(* CODESYS project AM402.project

Project tree, tasks and I/O mapping:
  Device : AM402-CPU1608TP/TN, Shenzhen Inovance Control Technology, version 3.5.11.11
    application Application
      libraries: Standard, * (System); SysTimeRtc, * (System); CmpHCMotion, 1.1.0.2 (Inovance); MemoryUtils, * (3S - Smart Software Solutions GmbH)
      task ETHERCAT (cyclic, interval 4000 µs, priority 0) calls ETHERCAT.EtherCAT_Task, MAIN
      program MAIN [ST]: io, motion, save_check, save_apply, supply, work, cut, cut_profile_update
      DataMain/
        data type HMIData
        data type SaveData
        data type SaveDataBig
        data type ProcessData
      DataWork/
        data type SupplyData
        data type WorkData
        data type CutData
        data type CutProfile
        data type CutProfileStep
      Enum/
        data type State
      Object/
        data type Button
        data type Cylinder
        data type AxisLinear
      function StateNext [ST]
      Symbols
      function block AxisLinearFB [ST]
    HardWare Configuration
    Network Configuration
      LocalBus Config
      EtherCAT Config
    Device Diagnosis
    Resources List
    ConfigStorage
    SoftMotion General Axis Pool
    HIGH_SPEED_IO : High Speed IO Module, Inovance, version 00.00.00.20
        unmapped channels: InputData, OutputData
      HSIO
    HwConfiguratioinDevice : SystemHardwareConfig, AM600 of Inovance, version 00.00.00.10
        settings: NetworkConfigArray.NetworkConfigArray.BusType = 10; NetworkConfigArray.NetworkConfigArray.RackSum = 1; NetworkConfigArray.NetworkConfigArray.HardwareConfigArray.HardwareConfigArray.RackNo = 1
    ETHERCAT : EtherCAT Master SoftMotion, 3S - Smart Software Solutions GmbH, version 3.5.11.10
        settings:  = 0; NetworkName = 'eth1'; SelectNetworkByName = TRUE; DisableTaskGeneration = True; SyncOffset = 20
      XINJE_DS5C1_CoE_Drive_Rev4_0 : XINJE-DS5C1 EtherCAT(CoE) Drive Rev4.0 v3.7.70, Xinje Electronics, Inc., order no. XINJE-DS5C1 CoE Drive Rev4.0, version Revision=16#20201207
          settings: StationAlias = 1; DC sync0 cycletime = 4000; DC sync1 cycletime = 4000; Interpolation time period.Value = 4
          unmapped channels: Control Word, TargetPosition, TargetVelocity, TargetTorque, ModeOfOperation, Status Word, ActualPosition, Velocity actual value, ActualTorque, ModeOfOperationDisplay
        Axis : Axis, 3S - Smart Software Solutions GmbH, order no. 0, version 4.0.0.0
            settings: wDriveID = 0; dwRatioTechUnitsDenom = 16384; iRatioTechUnitsNum = 625; eRampType = 3; ScalingIncs = 131072; ScalingUnits = 5000; AdrOffset_8010 = 2; BitOffset_8010 = 0; BitLength_8010 = 16; Address_8010 = '%QW1'; Type_8010 = 'UINT'; AddressPointer_8010 = ADR(%QW1); AdrOffset_8020 = 4; BitOffset_8020 = 0; BitLength_8020 = 32; Address_8020 = '%QD1'; Type_8020 = 'DINT'; AddressPointer_8020 = ADR(%QD1); AdrOffset_8030 = 8; BitOffset_8030 = 0; BitLength_8030 = 32; Address_8030 = '%QD2'; Type_8030 = 'DINT'; AddressPointer_8030 = ADR(%QD2); AdrOffset_8040 = 12; BitOffset_8040 = 0; BitLength_8040 = 16; Address_8040 = '%QW6'; Type_8040 = 'INT'; AddressPointer_8040 = ADR(%QW6); AdrOffset_8050 = 14; BitOffset_8050 = 0; BitLength_8050 = 8; Address_8050 = '%QB14'; Type_8050 = 'SINT'; AddressPointer_8050 = ADR(%QB14); AdrOffset_8060 = 4294967295; BitOffset_8060 = 0; BitLength_8060 = 0; Address_8060 = '';
              Type_8060 = ''; AddressPointer_8060 = 0; AdrOffset_8070 = 4294967295; BitOffset_8070 = 0; BitLength_8070 = 0; Address_8070 = ''; Type_8070 = ''; AddressPointer_8070 = 0; AdrOffset_8080 = 4294967295; BitOffset_8080 = 0; BitLength_8080 = 0; Address_8080 = ''; Type_8080 = ''; AddressPointer_8080 = 0; AdrOffset_8090 = 4294967295; BitOffset_8090 = 0; BitLength_8090 = 0; Address_8090 = ''; Type_8090 = ''; AddressPointer_8090 = 0; AdrOffset_8100 = 4294967295; BitOffset_8100 = 0; BitLength_8100 = 0; Address_8100 = ''; Type_8100 = ''; AddressPointer_8100 = 0; AdrOffset_8510 = 2; BitOffset_8510 = 0; BitLength_8510 = 16; Address_8510 = '%IW1'; Type_8510 = 'UINT'; AddressPointer_8510 = ADR(%IW1); AdrOffset_8520 = 4; BitOffset_8520 = 0; BitLength_8520 = 32; Address_8520 = '%ID1'; Type_8520 = 'DINT'; AddressPointer_8520 = ADR(%ID1); AdrOffset_8530 = 8; BitOffset_8530 = 0;
              BitLength_8530 = 32; Address_8530 = '%ID2'; Type_8530 = 'DINT'; AddressPointer_8530 = ADR(%ID2); AdrOffset_8540 = 12; BitOffset_8540 = 0; BitLength_8540 = 16; Address_8540 = '%IW6'; Type_8540 = 'INT'; AddressPointer_8540 = ADR(%IW6); AdrOffset_8550 = 14; BitOffset_8550 = 0; BitLength_8550 = 8; Address_8550 = '%IB14'; Type_8550 = 'SINT'; AddressPointer_8550 = ADR(%IB14); AdrOffset_8560 = 4294967295; BitOffset_8560 = 0; BitLength_8560 = 0; Address_8560 = ''; Type_8560 = ''; AddressPointer_8560 = 0; AdrOffset_8570 = 4294967295; BitOffset_8570 = 0; BitLength_8570 = 0; Address_8570 = ''; Type_8570 = ''; AddressPointer_8570 = 0; AdrOffset_8580 = 4294967295; BitOffset_8580 = 0; BitLength_8580 = 0; Address_8580 = ''; Type_8580 = ''; AddressPointer_8580 = 0; AdrOffset_8590 = 4294967295; BitOffset_8590 = 0; BitLength_8590 = 0; Address_8590 = ''; Type_8590 = ''; AddressPointer_8590 = 0;
              AdrOffset_8600 = 4294967295; BitOffset_8600 = 0; BitLength_8600 = 0; Address_8600 = ''; Type_8600 = ''; AddressPointer_8600 = 0; AdrOffset_8600 = 4294967295; BitOffset_8600 = 0; BitLength_8600 = 0; Address_8610 = ''; Type_8610 = ''; AddressPointer_8610 = 0; AdrOffset_8620 = 4294967295; BitOffset_8620 = 0; BitLength_8620 = 0; Address_8620 = ''; Type_8620 = ''; AddressPointer_8620 = 0
      XINJE_DS5C1_CoE_Drive_Rev4_0_1 : XINJE-DS5C1 EtherCAT(CoE) Drive Rev4.0 v3.7.70, Xinje Electronics, Inc., order no. XINJE-DS5C1 CoE Drive Rev4.0, version Revision=16#20201207
          settings: StationAlias = 1; DC sync0 cycletime = 4000; DC sync1 cycletime = 4000; Interpolation time period.Value = 4
          unmapped channels: Control Word, TargetPosition, TargetVelocity, TargetTorque, ModeOfOperation, Status Word, ActualPosition, Velocity actual value, ActualTorque, ModeOfOperationDisplay
        Axis_1 : Axis, 3S - Smart Software Solutions GmbH, order no. 0, version 4.0.0.0
            settings: dwRatioTechUnitsDenom = 16384; iRatioTechUnitsNum = -625; eRampType = 3; ScalingIncs = 131072; ScalingUnits = 5000; InvertDirection = TRUE; AdrOffset_8010 = 16; BitOffset_8010 = 0; BitLength_8010 = 16; Address_8010 = '%QW8'; Type_8010 = 'UINT'; AddressPointer_8010 = ADR(%QW8); AdrOffset_8020 = 20; BitOffset_8020 = 0; BitLength_8020 = 32; Address_8020 = '%QD5'; Type_8020 = 'DINT'; AddressPointer_8020 = ADR(%QD5); AdrOffset_8030 = 24; BitOffset_8030 = 0; BitLength_8030 = 32; Address_8030 = '%QD6'; Type_8030 = 'DINT'; AddressPointer_8030 = ADR(%QD6); AdrOffset_8040 = 28; BitOffset_8040 = 0; BitLength_8040 = 16; Address_8040 = '%QW14'; Type_8040 = 'INT'; AddressPointer_8040 = ADR(%QW14); AdrOffset_8050 = 30; BitOffset_8050 = 0; BitLength_8050 = 8; Address_8050 = '%QB30'; Type_8050 = 'SINT'; AddressPointer_8050 = ADR(%QB30); AdrOffset_8060 = 4294967295; BitOffset_8060 = 0; BitLength_8060 = 0; Address_8060 = '';
              Type_8060 = ''; AddressPointer_8060 = 0; AdrOffset_8070 = 4294967295; BitOffset_8070 = 0; BitLength_8070 = 0; Address_8070 = ''; Type_8070 = ''; AddressPointer_8070 = 0; AdrOffset_8080 = 4294967295; BitOffset_8080 = 0; BitLength_8080 = 0; Address_8080 = ''; Type_8080 = ''; AddressPointer_8080 = 0; AdrOffset_8090 = 4294967295; BitOffset_8090 = 0; BitLength_8090 = 0; Address_8090 = ''; Type_8090 = ''; AddressPointer_8090 = 0; AdrOffset_8100 = 4294967295; BitOffset_8100 = 0; BitLength_8100 = 0; Address_8100 = ''; Type_8100 = ''; AddressPointer_8100 = 0; AdrOffset_8510 = 16; BitOffset_8510 = 0; BitLength_8510 = 16; Address_8510 = '%IW8'; Type_8510 = 'UINT'; AddressPointer_8510 = ADR(%IW8); AdrOffset_8520 = 20; BitOffset_8520 = 0; BitLength_8520 = 32; Address_8520 = '%ID5'; Type_8520 = 'DINT'; AddressPointer_8520 = ADR(%ID5); AdrOffset_8530 = 24; BitOffset_8530 = 0;
              BitLength_8530 = 32; Address_8530 = '%ID6'; Type_8530 = 'DINT'; AddressPointer_8530 = ADR(%ID6); AdrOffset_8540 = 28; BitOffset_8540 = 0; BitLength_8540 = 16; Address_8540 = '%IW14'; Type_8540 = 'INT'; AddressPointer_8540 = ADR(%IW14); AdrOffset_8550 = 30; BitOffset_8550 = 0; BitLength_8550 = 8; Address_8550 = '%IB30'; Type_8550 = 'SINT'; AddressPointer_8550 = ADR(%IB30); AdrOffset_8560 = 4294967295; BitOffset_8560 = 0; BitLength_8560 = 0; Address_8560 = ''; Type_8560 = ''; AddressPointer_8560 = 0; AdrOffset_8570 = 4294967295; BitOffset_8570 = 0; BitLength_8570 = 0; Address_8570 = ''; Type_8570 = ''; AddressPointer_8570 = 0; AdrOffset_8580 = 4294967295; BitOffset_8580 = 0; BitLength_8580 = 0; Address_8580 = ''; Type_8580 = ''; AddressPointer_8580 = 0; AdrOffset_8590 = 4294967295; BitOffset_8590 = 0; BitLength_8590 = 0; Address_8590 = ''; Type_8590 = ''; AddressPointer_8590 = 0;
              AdrOffset_8600 = 4294967295; BitOffset_8600 = 0; BitLength_8600 = 0; Address_8600 = ''; Type_8600 = ''; AddressPointer_8600 = 0; AdrOffset_8600 = 4294967295; BitOffset_8600 = 0; BitLength_8600 = 0; Address_8610 = ''; Type_8610 = ''; AddressPointer_8610 = 0; AdrOffset_8620 = 4294967295; BitOffset_8620 = 0; BitLength_8620 = 0; Address_8620 = ''; Type_8620 = ''; AddressPointer_8620 = 0
  SMElement/
    SM0_SM511
    SM512_SM1023
    SM1024_SM1535
    SM1536_SM2047
    SM2048_SM2559
    SM2560_SM3071
    SM3072_SM3583
    SM3584_SM4095
    SM4096_SM4607
    SM4608_SM5119
    SM5120_SM5631
    SM5632_SM6143
    SM6144_SM6655
    SM6656_SM7167
    SM7168_SM7679
    SM7680_SM8191
    SM8192_SM8703
    SM8704_SM9215
    SM9216_SM9727
    SM9728_SM9999
  SDElement/
    SD0_SD511
    SD512_SD1023
    SD1024_SD1535
    SD1536_SD2047
    SD2048_SD2559
    SD2560_SD3071
    SD3072_SD3583
    SD3584_SD4095
    SD4096_SD4607
    SD4608_SD5119
    SD5120_SD5631
    SD5632_SD6143
    SD6144_SD6655
    SD6656_SD7167
    SD7168_SD7679
    SD7680_SD8191
    SD8192_SD8703
    SD8704_SD9215
    SD9216_SD9727
    SD9728_SD9999
*)

// Device/Application/DataMain/HMIData
{ attribute 'pack_mode' := ''}
TYPE HMIData :
STRUCT
	//
	save_data: SaveData;
	save: BOOL;
	save_need_check: BOOL;
	save_need: BOOL;
	//
	cut_profile_name_as_array: ARRAY[0..19] OF BYTE;
	cut_profile: CutProfile;
	cut_profile_points_x: ARRAY[0..(5*4-1+4)] OF UDINT;
	cut_profile_points_y: ARRAY[0..(5*4-1+4)] OF UDINT;
	cut_profile_point_count: UINT;
	cut_profile_bound_x: UDINT;
	cut_profile_bound_y: UDINT;
	cut_profile_index_changed: BOOL;
	cut_profile_list_update: BOOL;
	cut_profile_update: BOOL;
	//
	plc_ready: BOOL;
	hmi_ready: BOOL;
	run: BOOL;
	stop: BOOL;
	home: BOOL;
	manual_cut: BOOL;
	//
	supply_clamp_drag: BOOL;
	supply_clamp_hold: BOOL;
	supply_air_cool: BOOL;
	jog_micron_per_sec: UINT;
	jog_n: BOOL;
	jog_p: BOOL;
	jog_index: UINT;
	overload_resolved: BOOL;
	work_piece_count: UINT;
	//
	view_run: BOOL;
	view_stop: BOOL;
	view_air_ready: BOOL;
	view_can_run: BOOL;
	view_can_stop: BOOL;
	view_can_home: BOOL;
	//
	view_supply_position_micron: UDINT;
	view_supply_torque_mNm: UDINT;
	view_supply_foil_position_micron: UDINT;
	view_supply_sensor_hold: BOOL;
	view_supply_sensor_drag: BOOL;
	view_supply_foil_short: BOOL;
	view_cut_position_micron: UDINT;
	view_cut_torque_mNm: UDINT;
	view_cut_depth_micron: UDINT;
	view_work_piece_remain: UINT;
	//
	view_overload: BOOL;
	view_cycle_time_msec: UDINT;
	//
	view_state_work: INT;
	view_state_supply: INT;
	view_state_cut: INT;
END_STRUCT
END_TYPE

// Device/Application/DataMain/SaveData
{ attribute 'pack_mode' := ''}
TYPE SaveData :
STRUCT
	set_done: BOOL;
	//
	supply_ramp_time_msec: UINT;
	supply_jerk_factor: UINT;
	supply_hold_n_delay_msec: UINT;
	supply_hold_p_delay_msec: UINT;
	supply_drag_n_delay_msec: UINT;
	supply_drag_p_delay_msec: UINT;
	//
	cut_ramp_time_msec: UINT;
	cut_jerk_factor: UINT;
	cut_begin_micron: UDINT;
	//
	blade_thickness_micron: UINT; // độ dày lưỡi dao
	cut_depth_end_micron: UDINT; // độ sâu cắt đứt
	cut_retract_micron_per_sec: UDINT; // tốc độ lùi sau khi cắt
	cut_profile_index: UINT;
	manual_cut_micron_per_sec: UDINT; // tốc độ cắt thủ công
	//
	cut_profiles_name: ARRAY[0..9] OF STRING(20);
END_STRUCT
END_TYPE

// Device/Application/DataWork/SupplyData
{ attribute 'pack_mode' := ''}
TYPE SupplyData :
STRUCT
	state: INT;
	sensor_hold: BOOL;
	sensor_drag: BOOL;
	axis: AxisLinear;
	axis_fb: AxisLinearFB;
	clamp_drag: Cylinder;
	clamp_hold: Cylinder;
	air_cool: Cylinder;
	//
	foil_position_micron: LREAL;
	foil_position_target_micron: LREAL;
	foil_micron_per_sec: LREAL;
	foil_position_delta_micron: LREAL;
	foil_short: BOOL;
END_STRUCT
END_TYPE

// Device/Application/DataWork/WorkData
{ attribute 'pack_mode' := ''}
TYPE WorkData :
STRUCT
	state: INT;
	run: Button;
	run_timer: TON;
	can_run: BOOL;
	stop: Button;
	can_stop: BOOL;
	air_ready: BOOL;
	home: Button;
	can_home: BOOL;
	overload: Button;
	jog_i: POINTER TO AxisLinear;
	cut_profile: CutProfile;
	cut_profile_step_index: UINT;
	cut_profile_step: POINTER TO CutProfileStep;
	blade_thickness_micron: LREAL;
	cut_depth_end_micron: LREAL;
	work_piece_remain: UINT;
	manual_cut_clamp: BOOL;
	manual_cut_micron_per_sec: LREAL;
END_STRUCT
END_TYPE

// Device/Application/DataWork/CutData
{ attribute 'pack_mode' := ''}
TYPE CutData :
STRUCT
	state: INT;
	axis: AxisLinear;
	axis_fb: AxisLinearFB;
	blade_is_on: BOOL;
	//
	begin_micron: LREAL;
	depth_micron: LREAL;
	cut_micron_per_sec: LREAL;
	cut_retract_micron_per_sec: LREAL;
END_STRUCT
END_TYPE

// Device/Application/Enum/State
{attribute 'qualified_only'}
{attribute 'strict'}
TYPE State :
(
	NONE := 0,
	RST := 1,
	RST_DONE := 50,
	HOME := 51,
	HOME_FORWARD := 71,
	HOME_DONE := 90,
	HOME_OFFSET := 91,
	HOME_OFFSET_DONE := 99,
	READY := 100,
	RUN := 101,
	RUN_ING := 200
);
END_TYPE

// Device/Application/Object/Button
{ attribute 'pack_mode' := ''}
TYPE Button :
STRUCT
	on: BOOL;
	rise: R_TRIG;
	rise_physical: R_TRIG;
	fall: F_TRIG;
	fall_physical: F_TRIG;
END_STRUCT
END_TYPE

// Device/Application/Object/Cylinder
{ attribute 'pack_mode' := ''}
TYPE Cylinder :
STRUCT
	on: BOOL;
	n_timer: TON;
	p_timer: TON;
END_STRUCT
END_TYPE

// Device/Application/Object/AxisLinear
{ attribute 'pack_mode' := ''}
TYPE AxisLinear :
STRUCT
	///////
	//REF//
	///////
	ref: POINTER TO SM3_Drive_ETC_DS402_CyclicSync.AXIS_REF_ETC_DS402_CS;
	read_status: POINTER TO MC_ReadStatus;
	set_mode: POINTER TO SMC_SetControllerMode;
	limit_torque: POINTER TO MC_SetTorqueLimit;
	power: POINTER TO MC_Power;
	reset: POINTER TO MC_Reset;
	stop: POINTER TO MC_Stop;
	inch: POINTER TO SMC_Inch;
	sp: POINTER TO MC_SetPosition;
	mabs: POINTER TO MC_MoveAbsolute;
	////////
	//DATA//
	////////
	encoder_resolution: UDINT;
	torque_rated_Nm: LREAL;
	///////////
	//PROCESS//
	///////////
	state: INT;
	torque_Nm: LREAL;
	overload: BOOL;
	overload_timer: TON;
	//home
	home_done: BOOL; // = TRUE khi về gốc thành công, chỉ về gốc khi bật máy
	home_torque_Nm: LREAL;
	home_hit_timer: TON;
	home_offset_absolute_micron: LREAL; // vị trí từ điểm va chạm đến gốc tuyệt đối, xem hàm save_apply()
	home_back_micron_per_sec: LREAL; // tốc độ lùi về lấy gốc
	home_forward_micron_per_sec: LREAL; // tốc độ tiến sau khi lấy gốc xong
	home_offset_micron: LREAL; // giá trị này để thực hiện lệnh state = State.HOME_OFFSET ở trong AxisLinearFB
	//
	jog_micron_per_sec: LREAL; // tốc độ jog
	jog_direction: INT; // hướng jog
	max_micron: LREAL; // giới hạn vị trí tối đa có thể di chuyển từ gốc tuyệt đối
	max_micron_per_sec: LREAL; // giới hạn tốc độ tối đa
	ramp_time_sec: LREAL; // thời gian tăng, giảm tốc
	jerk_factor: LREAL; // độ giật, giá trị jerk của các hàm dịch chuyển sẽ bằng jerk := jerk_factor * acceleration
	//run
	target_position_micron: LREAL; // sử dụng cho state = State.RUN ở trong AxisLinearFB
	target_velocity_micron_per_sec: LREAL; // sử dụng cho state = State.RUN ở trong AxisLinearFB
END_STRUCT
END_TYPE

// Device/Application/DataWork/CutProfile
{ attribute 'pack_mode' := ''}
TYPE CutProfile :
STRUCT
	length_micron: UDINT;
	cut_micron_per_sec: UDINT;
	supply_micron_per_sec: UDINT;
	steps: ARRAY[0..4] OF CutProfileStep;
END_STRUCT
END_TYPE

// Device/Application/DataWork/CutProfileStep
{ attribute 'pack_mode' := ''}
TYPE CutProfileStep :
STRUCT
	active: BOOL;
	begin_micron: UDINT;
	width_micron: UDINT;
	depth_begin_micron: UDINT;
	depth_end_micron: UDINT;
END_STRUCT
END_TYPE

// Device/Application/DataMain/SaveDataBig
{ attribute 'pack_mode' := ''}
TYPE SaveDataBig :
STRUCT
	set_done: BOOL;
	//
	cut_profiles: ARRAY[0..9] OF CutProfile;
END_STRUCT
END_TYPE

// Device/Application/DataMain/ProcessData
{ attribute 'pack_mode' := ''}
TYPE ProcessData :
STRUCT
	cut_profile_name: STRING(20);
	cut_profile_name_changed: BOOL;
	cut_profile_changed: BOOL;
	cut_profile_list_update_need: BOOL;
	cut_profile_update_need: BOOL;
	supply_foil_short_rise: R_TRIG;
END_STRUCT
END_TYPE

// Device/Application/MAIN
PROGRAM MAIN
VAR
	RTC_last: ULINT;
	RTC : ULINT;
	//
	axiss: ARRAY [0..1] OF POINTER TO SM3_Drive_ETC_DS402_CyclicSync.AXIS_REF_ETC_DS402_CS;
	// dùng pointer để dễ dàng thao tác với nhiều trục hơn, xem hàm motion()
	axiss_read: ARRAY[0..1] OF SMC3_ETC_ReadParameter_CoE;
	axiss_read_status: ARRAY[0..1] OF MC_ReadStatus;
	axiss_set_mode: ARRAY[0..1] OF SMC_SetControllerMode;
	axiss_limit_torque: ARRAY[0..1] OF MC_SetTorqueLimit; // không có sẵn, cần cài thư viện CmpHCMotion của Inovance, PLC khác có thể khác
	axiss_power: ARRAY[0..1] OF MC_Power; // bật tắt động cơ
	axiss_reset: ARRAY[0..1] OF MC_Reset; // reset lỗi
	axiss_stop: ARRAY[0..1] OF MC_Stop; // dừng
	axiss_inch: ARRAY[0..1] OF SMC_Inch;
	axiss_sp: ARRAY[0..1] OF MC_SetPosition;
	axiss_mabs: ARRAY[0..1] OF MC_MoveAbsolute;
	axiss_encoder_resolution: ARRAY[0..1] OF UDINT;
	axiss_rated_torque_Nm: ARRAY[0..1] OF LREAL;
	axiss_ready: BOOL;
	//
	state_main: INT;
	main_save: Button;
	supply_data: SupplyData;
	cut_data: CutData;
	work_data: WorkData;
	hmi_data: HMIData;
	process_data: ProcessData;
	//
	i: UINT;
	j: UINT;
	k: UINT;
	axis_linear_i: POINTER TO AxisLinear;
	axis_linear_fb_i: POINTER TO AxisLinearFB;
	cut_profile_i: POINTER TO CutProfile;
	cut_profile_step_i: POINTER TO CutProfileStep;
	//
	udint_min: UDINT;
	udint_max: UDINT;
END_VAR

VAR CONSTANT
	c_axis_count: UINT := 2;
	c_axis_i_max: UINT := c_axis_count - 1;
	c_cut_profile_count: UINT := 10;
	c_cut_profile_i_max: UINT := c_cut_profile_count - 1;
	c_cut_profile_step_count: UINT := 5;
	c_cut_profile_step_i_max: UINT := c_cut_profile_step_count - 1;
	c_name_length: UINT := 20;
	c_supply_travel_micron_max: UDINT := 289_000;
	c_supply_travel_micron_per_sec_max: LREAL := (3000 / 60) * 5_000; // 3000 rpm, 5_000 micron 1 vòng
	c_cut_depth_micron_max: UDINT := 155_000;
	c_cut_travel_micron_per_sec_max: LREAL := (3000 / 60) * 5_000; // 3000 rpm, 5_000 micron 1 vòng
	c_cut_begin_micron_max: UDINT := 80_000;
END_VAR

VAR RETAIN
	save_data: SaveData;
	save_data_big: SaveDataBig;
END_VAR

SysTimeRtc.SysTimeRtcHighResGet(pTimestamp:= RTC);
IF state_main > 10 THEN
	motion();
	// chạy hàm motion(), vì state 11 trở đi có đoạn đọc dữ liệu của Servo
	// mà hàm motion() này lại bao gồm tất cả các lệnh của Servo
	// có thể thay đổi logic đoạn này nhưng không cần thiết lắm
END_IF

CASE state_main OF
	State.NONE: // khi khởi động thì state_main = 0 tức là = State.NONE
		axiss[0] := ADR(Axis_1); // k = ADR(x) viết tắt cho "address of x" là hàm để lấy giá trị con trỏ (pointer) về biến x
		axiss[1] := ADR(Axis); // ví dụ muốn thay đổi giá trị của x ta sẽ viết k^ = 12345
		StateNext(state_main); // chuyển tới trạng thái tiếp theo
	1:
		FOR i := 0 TO c_axis_i_max BY 1 DO // hàm FOR, FOR i = 0 TO 3 BY 1 DO sẽ chạy 4 lần i = [0, 1, 2, 3]
			CASE i OF // hàm CASE, lựa chọn theo giá trị i
				0:
					axis_linear_i := ADR(cut_data.axis);
					axis_linear_fb_i := ADR(cut_data.axis_fb);
				1:
					axis_linear_i := ADR(supply_data.axis);
					axis_linear_fb_i := ADR(supply_data.axis_fb);
			END_CASE
			axis_linear_i^.ref := axiss[i];
			axis_linear_i^.read_status := ADR(axiss_read_status[i]);
			axis_linear_i^.set_mode := ADR(axiss_set_mode[i]);
			axis_linear_i^.limit_torque := ADR(axiss_limit_torque[i]);
			axis_linear_i^.power := ADR(axiss_power[i]);
			axis_linear_i^.reset := ADR(axiss_reset[i]);
			axis_linear_i^.stop := ADR(axiss_stop[i]);
			axis_linear_i^.inch := ADR(axiss_inch[i]);
			axis_linear_i^.sp := ADR(axiss_sp[i]);
			axis_linear_i^.mabs := ADR(axiss_mabs[i]);
			axis_linear_fb_i^.data := axis_linear_i;
		END_FOR
		StateNext(state_main);
	2:
		axiss_ready := TRUE; // biến tạm thời để kiểm tra tất cả các servo đã hoàn thành lệnh hay chưa
		FOR i := 0 TO c_axis_i_max BY 1 DO
			IF axiss[i]^.wCommunicationState <> 100 THEN
				// nếu trạng thái wCommunicationState của servo bất kỳ không = 100 thì
				// chứng tỏ chưa hoàn thành kết nối tất cả các servo, nên ta cho giá trị axiss_ready := FALSE
				axiss_ready := FALSE;
			END_IF
		END_FOR
		IF axiss_ready THEN // hoàn thành kết nối tất cả servo, ta đên bước tiếp theo
			state_main := 11;
		END_IF
	11:
		FOR i := 0 TO c_axis_i_max BY 1 DO
			// bật động cơ, phải đặt ba biến của hàm MC_Power này = TRUE
			axiss_power[i].Enable := TRUE;
			axiss_power[i].bDriveStart := TRUE;
			axiss_power[i].bRegulatorOn := TRUE;
		END_FOR
		StateNext(state_main);
	12:
		axiss_ready := TRUE;
		FOR i := 0 TO c_axis_i_max BY 1 DO
			IF NOT axiss_power[i].Status THEN // axiss_power[i].Status = TRUE tức là đã bật Servo thành công
				axiss_ready := FALSE;
			END_IF
		END_FOR
		IF axiss_ready THEN
			StateNext(state_main);
		END_IF
	13: // đọc dữ liệu từ servo
		FOR i := 0 TO c_axis_i_max BY 1 DO
			axiss_read[i].uiIndex := 16#608F; // mở ETHERCAT/XINJE_DS5C1.../ xem trong mục "CoE Online"
			axiss_read[i].usiSubIndex := 1; //
			axiss_read[i].xExecute := TRUE;
		END_FOR
		StateNext(state_main);
	14:
		axiss_ready := TRUE;
		FOR i := 0 TO c_axis_i_max BY 1 DO
			IF NOT axiss_read[i].xDone THEN
				axiss_ready := FALSE;
			END_IF
		END_FOR
		IF axiss_ready THEN
			FOR i := 0 TO c_axis_i_max BY 1 DO
				axiss_read[i].xExecute := FALSE;
				// Sau thực hiện hàm thành công phải đặt Execute = FALSE để cho lần đọc tiếp theo
				// vì đa số hàm chỉ chạy khi Execute chuyển từ FALSE sang TRUE (Rising edge)
				// xem Defination của hàm đê biết thêm chi tiết
				axiss_encoder_resolution[i] := DWORD_TO_UDINT(axiss_read[i].dwValue);
			END_FOR
			StateNext(state_main);
		END_IF
	15:
		FOR i := 0 TO c_axis_i_max BY 1 DO
			axiss_read[i].uiIndex := 16#6076;
			axiss_read[i].usiSubIndex := 0;
			axiss_read[i].xExecute := TRUE;
		END_FOR
		StateNext(state_main);
	16:
		axiss_ready := TRUE;
		FOR i := 0 TO c_axis_i_max BY 1 DO
			IF NOT axiss_read[i].xDone THEN
				axiss_ready := FALSE;
			END_IF
		END_FOR
		IF axiss_ready THEN
			FOR i := 0 TO c_axis_i_max BY 1 DO
				axiss_read[i].xExecute := FALSE;
				axiss_rated_torque_Nm[i] := DWORD_TO_LREAL(axiss_read[i].dwValue) * 1E-3;
			END_FOR
			StateNext(state_main);
		END_IF
	17:
		supply_data.axis.encoder_resolution := axiss_encoder_resolution[0];
		supply_data.axis.torque_rated_Nm := axiss_rated_torque_Nm[0];
		cut_data.axis.encoder_resolution := axiss_encoder_resolution[1];
		cut_data.axis.torque_rated_Nm := axiss_rated_torque_Nm[1];
		IF NOT save_data.set_done THEN
			save_data.set_done := TRUE;
			// biến "set_done" này nằm trong cấu trúc "save_data" nhằm mục đích
			// gán giá trị đầu cho biến lưu, đảm bảo đoạn gán dữ liệu này chỉ chạy 1 lần khi
			// PLC chạy lần dầu sau khi nạp lại chương trình.
			//
			save_data.supply_ramp_time_msec := 0_100;
			save_data.supply_jerk_factor := 10;
			save_data.supply_hold_n_delay_msec := 0_600;
			save_data.supply_hold_p_delay_msec := 0_700;
			save_data.supply_drag_n_delay_msec := 0_800;
			save_data.supply_drag_p_delay_msec := 0_900;
			//
			save_data.cut_ramp_time_msec := 0_100;
			save_data.cut_jerk_factor := 10;
			save_data.cut_begin_micron := 15_000;
			//
			save_data.blade_thickness_micron := 4_250;
			save_data.cut_depth_end_micron := 70_000;
			save_data.cut_retract_micron_per_sec := 25_000;
			save_data.cut_profile_index := 0;
			save_data.manual_cut_micron_per_sec := 15_000;
			FOR i := 0 TO c_cut_profile_i_max BY 1 DO
				save_data.cut_profiles_name[i] := CONCAT('Profile ', UINT_TO_STRING(i));
				// CONCAT là hàm nối 2 STRING với nhau
			END_FOR
		END_IF
		IF NOT save_data_big.set_done THEN
			save_data_big.set_done := TRUE;
			//
			FOR i := 0 TO c_cut_profile_i_max BY 1 DO
				cut_profile_i := ADR(save_data_big.cut_profiles[i]);
				cut_profile_i^.length_micron := 200_000;
				cut_profile_i^.cut_micron_per_sec := save_data.manual_cut_micron_per_sec;
				cut_profile_i^.supply_micron_per_sec := 100_000;
				FOR j := 0 TO c_cut_profile_step_i_max BY 1 DO
					cut_profile_step_i := ADR(cut_profile_i^.steps[j]);
					cut_profile_step_i^.active := TRUE;
					cut_profile_step_i^.begin_micron := 25_000 * (j + 1) + i;
					cut_profile_step_i^.width_micron := save_data.blade_thickness_micron * (j + 1) + i;
					cut_profile_step_i^.depth_begin_micron := 5_000 * (j + 1) + i * 5_000;
					cut_profile_step_i^.depth_end_micron := 10_000 * (j + 1);
				END_FOR
			END_FOR
		END_IF
		StateNext(state_main);
	18:
		process_data.cut_profile_name := save_data.cut_profiles_name[save_data.cut_profile_index];
		MEMUtils.MemCpy(
			ADR(hmi_data.cut_profile_name_as_array),
			ADR(process_data.cut_profile_name),
			UINT_TO_DWORD(c_name_length)
		);
		save_apply();
		process_data.cut_profile_list_update_need := TRUE; // cần cập nhật danh sách cut_profile
		process_data.cut_profile_update_need := TRUE;
		cut_profile_update();
		StateNext(state_main);
	19:
		hmi_data.plc_ready := TRUE; // sau khi đã khởi động Servo bla bla thì ta PLC ready
		work_data.state := State.RST; // reset work
		state_main := State.RUN_ING; // bước vào giai đoạn chạy
	State.RUN_ING:
		io(); // kiểm tra io (gồm PLC io và HMI)
		supply(); // hàm điều khiển cơ cấu cấp phôi (gồm servo và các xylanh khí nén)
		cut(); // hàm điều khiển trục cắt
		work(); // hàm phối hợp giữa cấp phôi và cắt
END_CASE

ACTION io:
////////////
//HMI DOWN//
///////////
IF hmi_data.hmi_ready THEN
	////////
	//WORK//
	////////
	work_data.run.rise(CLK:= hmi_data.run, Q=> );
	work_data.stop.rise(CLK:= hmi_data.stop, Q=> );
	work_data.home.rise(CLK:= hmi_data.home, Q=> );
	IF work_data.home.rise.Q AND work_data.can_home THEN
		supply_data.axis.home_done := FALSE;
		cut_data.axis.home_done := FALSE;
		work_data.state := State.HOME;
	END_IF
	work_data.overload.rise(CLK:= hmi_data.overload_resolved, Q=> );
	IF work_data.overload.rise.Q THEN
		work_data.overload.on := FALSE;
	END_IF
	//////////
	//SUPPLY//
	//////////
	IF work_data.state = State.RST_DONE OR work_data.state = State.READY THEN
		IF NOT hmi_data.manual_cut THEN
			supply_data.clamp_hold.on := hmi_data.supply_clamp_hold;
			supply_data.clamp_drag.on := hmi_data.supply_clamp_drag;
		END_IF
		supply_data.air_cool.on := hmi_data.supply_air_cool;
	ELSE
		hmi_data.supply_clamp_hold := supply_data.clamp_hold.on;
		hmi_data.supply_clamp_drag := supply_data.clamp_drag.on;
		hmi_data.supply_air_cool := supply_data.air_cool.on;
	END_IF
	////////
	//SAVE//
	////////
	IF hmi_data.save_need_check THEN
		save_check();
		hmi_data.save_need_check := FALSE;
	END_IF
	main_save.rise(CLK:= hmi_data.save, Q=> ); // Trên HMI sẽ xuất hiện nút save khi biến hmi_data.save_need = true.
	IF main_save.rise.Q THEN
		save_data := hmi_data.save_data;
		save_apply();
		hmi_data.save_need := FALSE;
		hmi_data.save := FALSE;
	END_IF
END_IF
/////////
//INPUT//
/////////
work_data.can_run := work_data.stop.fall_physical.CLK AND work_data.air_ready AND work_data.state = State.READY AND cut_data.blade_is_on;
work_data.can_stop := work_data.state >= State.NONE;
work_data.can_home := work_data.state = State.RST_DONE OR work_data.state = State.READY;
//
work_data.run.rise_physical(CLK:= %IX0.4, Q=> );
work_data.stop.fall_physical(CLK:= %IX0.5, Q=> );
work_data.manual_cut_clamp := %IX0.6;
work_data.air_ready := %IX0.7;
supply_data.sensor_hold := %IX1.0;
supply_data.sensor_drag := %IX1.1;
cut_data.blade_is_on := %IX1.2;
work_data.overload.rise(CLK:= work_data.overload.on, Q=> );
work_data.run_timer(IN:= work_data.run.rise.CLK OR work_data.run.rise_physical.CLK, PT:= , Q=> , ET=> );
IF work_data.stop.fall_physical.CLK THEN
	CASE work_data.state OF
		State.RST_DONE:
			IF work_data.run.rise.Q OR work_data.run.rise_physical.Q THEN
				work_data.state := State.HOME;
			END_IF
		State.READY:
			IF hmi_data.manual_cut THEN
				supply_data.clamp_hold.on := work_data.manual_cut_clamp;
				supply_data.clamp_drag.on := work_data.manual_cut_clamp;
				hmi_data.supply_clamp_hold := supply_data.clamp_hold.on;
				hmi_data.supply_clamp_drag := supply_data.clamp_drag.on;
				IF work_data.can_run AND work_data.run_timer.Q THEN
					work_data.state := 171;
				END_IF
			ELSIF work_data.can_run AND (work_data.run.rise.Q OR work_data.run.rise_physical.Q) THEN
				hmi_data.work_piece_count := MAX(1, hmi_data.work_piece_count);
				work_data.work_piece_remain := hmi_data.work_piece_count;
				work_data.state := State.RUN;
			END_IF
	END_CASE
END_IF
IF (work_data.stop.rise.Q OR work_data.stop.fall_physical.Q OR work_data.overload.rise.Q) AND work_data.can_stop THEN
	work_data.state := State.RST;
END_IF
//
supply_data.clamp_drag.n_timer(IN:= NOT supply_data.clamp_drag.on, PT:= , Q=> , ET=> );
supply_data.clamp_drag.p_timer(IN:= supply_data.clamp_drag.on, PT:= , Q=> , ET=> );
supply_data.clamp_hold.n_timer(IN:= NOT supply_data.clamp_hold.on, PT:= , Q=> , ET=> );
supply_data.clamp_hold.p_timer(IN:= supply_data.clamp_hold.on, PT:= , Q=> , ET=> );
//////////
//OUTPUT//
//////////
%QX0.0 := supply_data.clamp_drag.on;
%QX0.1 := supply_data.clamp_hold.on;
%QX0.2 := supply_data.air_cool.on;
//////////
//HMI UP//
//////////
IF hmi_data.hmi_ready THEN
	hmi_data.view_run := work_data.run.rise_physical.CLK;
	hmi_data.view_stop := work_data.stop.fall_physical.CLK;
	hmi_data.view_air_ready := work_data.air_ready;
	hmi_data.view_can_run := work_data.can_run;
	hmi_data.view_can_stop := work_data.can_stop;
	hmi_data.view_can_home := work_data.can_home;
	hmi_data.view_overload := work_data.overload.on;
	//
	hmi_data.view_supply_position_micron := LREAL_TO_UDINT(supply_data.axis.ref^.fActPosition);
	hmi_data.view_supply_torque_mNm := LREAL_TO_UDINT(ABS(supply_data.axis.torque_Nm) * 1E3);
	hmi_data.view_supply_foil_position_micron := LREAL_TO_UDINT(supply_data.foil_position_micron);
	hmi_data.view_supply_sensor_hold := supply_data.sensor_hold;
	hmi_data.view_supply_sensor_drag := supply_data.sensor_drag;
	// hàm R_TRIG (rising edge detect), khi supply_data.foil_short chuyển từ FALSE -> TRUE
	// kích hoạt biến view_supply_foil_short để hiển thị nút hết phôi trên HMI
	process_data.supply_foil_short_rise(CLK:= supply_data.foil_short, Q=> );
	IF process_data.supply_foil_short_rise.Q THEN
		hmi_data.view_supply_foil_short := TRUE;
	END_IF
	hmi_data.view_cut_position_micron := LREAL_TO_UDINT(cut_data.axis.ref^.fActPosition);
	hmi_data.view_cut_torque_mNm := LREAL_TO_UDINT(ABS(cut_data.axis.torque_Nm) * 1E3);
	hmi_data.view_cut_depth_micron := LREAL_TO_UDINT(cut_data.axis.mabs^.Position - cut_data.begin_micron);
	hmi_data.view_work_piece_remain := work_data.work_piece_remain;
	//
	hmi_data.view_state_work := work_data.state;
	hmi_data.view_state_supply := supply_data.state;
	hmi_data.view_state_cut := cut_data.state;
	// cập nhật khi chọn cut_profile trên HMI
	// HMI sẽ set hmi_data.cut_profile_index_changed := TRUE khi chọn cut_profile
	IF hmi_data.cut_profile_index_changed THEN
		hmi_data.cut_profile_index_changed := FALSE;
		hmi_data.save_need_check := TRUE;
		process_data.cut_profile_update_need := TRUE;
	END_IF
	IF process_data.cut_profile_update_need AND NOT hmi_data.cut_profile_update THEN
		process_data.cut_profile_update_need := FALSE;
		cut_profile_update();
		hmi_data.cut_profile_update := TRUE; // cập nhật cut_profile trên HMI khi cần cập nhật và đang không cập nhật 
	END_IF
	IF process_data.cut_profile_list_update_need AND NOT hmi_data.cut_profile_list_update THEN
		process_data.cut_profile_list_update_need := FALSE;
		hmi_data.cut_profile_list_update := TRUE; // cập nhật cut_profile_list trên HMI khi cần cập nhật và đang không cập nhật
	END_IF
END_IF
END_ACTION

ACTION motion:
FOR i := 0 TO c_axis_i_max BY 1 DO
	axiss_read[i](
		xExecute:= , 
		xAbort:= , 
		uiIndex:= , 
		usiSubIndex:= , 
		Axis:= axiss[i]^, 
		xDone=> , 
		xBusy=> , 
		xError=> , 
		usiDataLength=> , 
		dwValue=> , 
		dwErrorCode=> , 
		eError=> );
	axiss_read_status[i](
		Axis:= axiss[i]^, 
		Enable:= , 
		Valid=> , 
		Busy=> , 
		Error=> , 
		ErrorID=> , 
		Disabled=> , 
		Errorstop=> , 
		Stopping=> , 
		StandStill=> , 
		DiscreteMotion=> , 
		ContinuousMotion=> , 
		SynchronizedMotion=> , 
		Homing=> , 
		ConstantVelocity=> , 
		Accelerating=> , 
		Decelerating=> , 
		FBErrorOccured=> );
	axiss_set_mode[i](
		Axis:= axiss[i]^, 
		bExecute:= , 
		nControllerMode:= , 
		bDone=> , 
		bBusy=> , 
		bError=> , 
		nErrorID=> );
	axiss_limit_torque[i](
		Axis:= axiss[i]^, 
		Execute:= , 
		PositiveEnable:= , 
		PositiveValue:= , 
		NegativeEnable:= , 
		NegativeValue:= , 
		Done=> , 
		Busy=> , 
		Error=> , 
		ErrorID=> );
	axiss_power[i](
		Axis:= axiss[i]^,
		Enable:= , 
		bRegulatorOn:= , 
		bDriveStart:= , 
		Status=> , 
		bRegulatorRealState=> , 
		bDriveStartRealState=> , 
		Busy=> , 
		Error=> , 
		ErrorID=> );
	axiss_reset[i](
		Axis:= axiss[i]^,
		Execute:= ,
		Done=> ,
		Busy=> ,
		Error=> ,
		ErrorID=> );
	axiss_stop[i](
		Axis:= axiss[i]^, 
		Execute:= , 
		Deceleration:= , 
		Jerk:= , 
		Done=> , 
		Busy=> , 
		Error=> , 
		ErrorID=> );
	axiss_inch[i](
		Axis:= axiss[i]^, 
		InchForward:= , 
		InchBackward:= , 
		Distance:= , 
		Velocity:= , 
		Acceleration:= , 
		Deceleration:= , 
		Jerk:= , 
		Busy=> , 
		CommandAborted=> , 
		Error=> , 
		ErrorId=> );
	axiss_sp[i](
		Axis:= axiss[i]^, 
		Execute:= , 
		Position:= , 
		Mode:= , 
		Done=> , 
		Busy=> , 
		Error=> , 
		ErrorID=> );
	axiss_mabs[i](
		Axis:= axiss[i]^, 
		Execute:= , 
		Position:= , 
		Velocity:= , 
		Acceleration:= , 
		Deceleration:= , 
		Jerk:= , 
		Direction:= , 
		BufferMode:= , 
		Done=> , 
		Busy=> , 
		Active=> , 
		CommandAborted=> , 
		Error=> , 
		ErrorID=> );
END_FOR
END_ACTION

ACTION save_check:
MEMUtils.MemCpy( // cần cài đặt thư viện MEMUtils để sử dụng hàm này
	ADR(process_data.cut_profile_name),
	ADR(hmi_data.cut_profile_name_as_array),
	UINT_TO_DWORD(c_name_length)
);
process_data.cut_profile_name_changed := save_data.cut_profiles_name[hmi_data.save_data.cut_profile_index] <> process_data.cut_profile_name;

cut_profile_i := ADR(save_data_big.cut_profiles[hmi_data.save_data.cut_profile_index]);
process_data.cut_profile_changed := (
	cut_profile_i^.length_micron <> hmi_data.cut_profile.length_micron OR
	cut_profile_i^.cut_micron_per_sec <> hmi_data.cut_profile.cut_micron_per_sec OR
	cut_profile_i^.supply_micron_per_sec <> hmi_data.cut_profile.supply_micron_per_sec
);
FOR i := 0 TO c_cut_profile_step_i_max BY 1 DO
	process_data.cut_profile_changed := (
		process_data.cut_profile_changed OR
		cut_profile_i^.steps[i].active <> hmi_data.cut_profile.steps[i].active OR
		cut_profile_i^.steps[i].begin_micron <> hmi_data.cut_profile.steps[i].begin_micron OR
		cut_profile_i^.steps[i].width_micron <> hmi_data.cut_profile.steps[i].width_micron OR
		cut_profile_i^.steps[i].depth_begin_micron <> hmi_data.cut_profile.steps[i].depth_begin_micron OR
		cut_profile_i^.steps[i].depth_end_micron <> hmi_data.cut_profile.steps[i].depth_end_micron
	);
END_FOR

hmi_data.save_need := (
	save_data.supply_ramp_time_msec <> hmi_data.save_data.supply_ramp_time_msec OR
	save_data.supply_jerk_factor <> hmi_data.save_data.supply_jerk_factor OR
	save_data.supply_hold_n_delay_msec <> hmi_data.save_data.supply_hold_n_delay_msec OR
	save_data.supply_hold_p_delay_msec <> hmi_data.save_data.supply_hold_p_delay_msec OR
	save_data.supply_drag_n_delay_msec <> hmi_data.save_data.supply_drag_n_delay_msec OR
	save_data.supply_drag_p_delay_msec <> hmi_data.save_data.supply_drag_p_delay_msec OR
	//
	save_data.cut_ramp_time_msec <> hmi_data.save_data.cut_ramp_time_msec OR
	save_data.cut_jerk_factor <> hmi_data.save_data.cut_jerk_factor OR
	save_data.cut_begin_micron <> hmi_data.save_data.cut_begin_micron OR
	//
	save_data.blade_thickness_micron <> hmi_data.save_data.blade_thickness_micron OR
	save_data.cut_depth_end_micron <> hmi_data.save_data.cut_depth_end_micron OR
	save_data.cut_retract_micron_per_sec <> hmi_data.save_data.cut_retract_micron_per_sec OR
	save_data.cut_profile_index <> hmi_data.save_data.cut_profile_index OR
	save_data.manual_cut_micron_per_sec <> hmi_data.save_data.manual_cut_micron_per_sec OR
	//
	process_data.cut_profile_name_changed OR
	process_data.cut_profile_changed
);
END_ACTION

ACTION save_apply:
/////////
//LIMIT//
/////////
save_data.supply_ramp_time_msec := MAX(0_100, MIN(1_000, save_data.supply_ramp_time_msec));
save_data.supply_jerk_factor := MAX(10, MIN(50, save_data.supply_jerk_factor));
save_data.supply_hold_n_delay_msec := MAX(0_100, MIN(5_000, save_data.supply_hold_n_delay_msec));
save_data.supply_hold_p_delay_msec := MAX(0_100, MIN(5_000, save_data.supply_hold_p_delay_msec));
save_data.supply_drag_n_delay_msec := MAX(0_100, MIN(5_000, save_data.supply_drag_n_delay_msec));
save_data.supply_drag_p_delay_msec := MAX(0_100, MIN(5_000, save_data.supply_drag_p_delay_msec));
//
save_data.cut_ramp_time_msec := MAX(0_100, MIN(1_000, save_data.cut_ramp_time_msec));
save_data.cut_jerk_factor := MAX(10, MIN(50, save_data.cut_jerk_factor));
save_data.cut_begin_micron := MIN(c_cut_begin_micron_max, save_data.cut_begin_micron);
//
save_data.blade_thickness_micron := MAX(1_000, MIN(10_000, save_data.blade_thickness_micron));
save_data.cut_depth_end_micron := MAX(1_000, MIN(c_cut_depth_micron_max, save_data.cut_depth_end_micron));
save_data.cut_retract_micron_per_sec := MAX(1_000, MIN(150_000, save_data.cut_retract_micron_per_sec));
save_data.cut_profile_index := MAX(0, MIN(c_cut_profile_i_max, save_data.cut_profile_index));
save_data.manual_cut_micron_per_sec := MAX(1_000, MIN(150_000, save_data.manual_cut_micron_per_sec));
//
IF process_data.cut_profile_name_changed THEN
	MEMUtils.MemCpy(
		ADR(process_data.cut_profile_name),
		ADR(hmi_data.cut_profile_name_as_array),
		UINT_TO_DWORD(c_name_length)
	);
	save_data.cut_profiles_name[save_data.cut_profile_index] := process_data.cut_profile_name;
	process_data.cut_profile_list_update_need := TRUE;
END_IF
IF process_data.cut_profile_changed THEN // cut_profile đã thay đổi ở save_check()
	hmi_data.cut_profile.cut_micron_per_sec := MAX(1_000, MIN(150_000, hmi_data.cut_profile.cut_micron_per_sec));
	hmi_data.cut_profile.supply_micron_per_sec := MAX(10_000, MIN(250_000, hmi_data.cut_profile.supply_micron_per_sec));
	FOR i := 0 TO c_cut_profile_step_i_max BY 1 DO
		cut_profile_step_i := ADR(hmi_data.cut_profile.steps[i]);
		cut_profile_step_i^.begin_micron := MAX(save_data.blade_thickness_micron, MIN(hmi_data.cut_profile.length_micron, cut_profile_step_i^.begin_micron));
		cut_profile_step_i^.width_micron := MAX(save_data.blade_thickness_micron, MIN(hmi_data.cut_profile.length_micron, cut_profile_step_i^.width_micron));
		cut_profile_step_i^.depth_begin_micron := MIN(c_cut_depth_micron_max, cut_profile_step_i^.depth_begin_micron);
		cut_profile_step_i^.depth_end_micron := MIN(c_cut_depth_micron_max, cut_profile_step_i^.depth_end_micron);
	END_FOR
	save_data_big.cut_profiles[save_data.cut_profile_index] := hmi_data.cut_profile;
	process_data.cut_profile_update_need := TRUE; // cần phải cập nhật cut_profile ở io()
END_IF
/////////
//APPLY//
/////////
supply_data.axis.home_hit_timer.PT := INT_TO_TIME(1_000);
supply_data.axis.home_offset_absolute_micron := 1_000;
supply_data.axis.home_back_micron_per_sec := 10_000;
supply_data.axis.home_forward_micron_per_sec := 30_000;
supply_data.axis.max_micron := UDINT_TO_LREAL(c_supply_travel_micron_max);
supply_data.axis.max_micron_per_sec := c_supply_travel_micron_per_sec_max;
supply_data.axis.ramp_time_sec := UINT_TO_LREAL(save_data.supply_ramp_time_msec) * 1E-3;
supply_data.axis.jerk_factor := UINT_TO_LREAL(save_data.supply_jerk_factor);
supply_data.axis.overload_timer.PT := INT_TO_TIME(1_000);
//
cut_data.axis.home_hit_timer.PT := INT_TO_TIME(1_000);
cut_data.axis.home_offset_absolute_micron := 1_000;
cut_data.axis.home_back_micron_per_sec := 10_000;
cut_data.axis.home_forward_micron_per_sec := 30_000;
cut_data.axis.max_micron := UDINT_TO_LREAL(c_cut_depth_micron_max);
cut_data.axis.max_micron_per_sec := c_cut_travel_micron_per_sec_max;
cut_data.axis.ramp_time_sec := UINT_TO_LREAL(save_data.cut_ramp_time_msec) * 1E-3;
cut_data.axis.jerk_factor := UINT_TO_LREAL(save_data.cut_jerk_factor);
cut_data.axis.overload_timer.PT := INT_TO_TIME(1_000);
cut_data.begin_micron := UDINT_TO_LREAL(save_data.cut_begin_micron);
cut_data.cut_retract_micron_per_sec := UDINT_TO_LREAL(save_data.cut_retract_micron_per_sec);
//
supply_data.clamp_hold.n_timer.PT := UINT_TO_TIME(save_data.supply_hold_n_delay_msec);
supply_data.clamp_hold.p_timer.PT := UINT_TO_TIME(save_data.supply_hold_p_delay_msec);
supply_data.clamp_drag.n_timer.PT := UINT_TO_TIME(save_data.supply_drag_n_delay_msec);
supply_data.clamp_drag.p_timer.PT := UINT_TO_TIME(save_data.supply_drag_p_delay_msec);
//
work_data.run_timer.PT := INT_TO_TIME(0_500);
work_data.blade_thickness_micron := UINT_TO_LREAL(save_data.blade_thickness_micron);
work_data.cut_depth_end_micron := UDINT_TO_LREAL(save_data.cut_depth_end_micron);
work_data.manual_cut_micron_per_sec := UDINT_TO_LREAL(save_data.manual_cut_micron_per_sec);
/////////
//FINAL//
/////////
hmi_data.save_data := save_data;
END_ACTION

ACTION supply:
////////
//MAIN//
////////
supply_data.axis_fb(data:= ); // data của hàm này đã được set ở hàm MAIN
CASE supply_data.state OF
	//////\\
	////\\\\
	//\\\\\\
	State.RST:
		supply_data.axis.state := State.RST;
		StateNext(supply_data.state);
	2:
		IF supply_data.axis.state = State.RST_DONE THEN
			supply_data.state := State.RST_DONE;
		END_IF
	//////\\
	////\\\\
	//\\\\\\
	State.HOME:
		supply_data.axis.state := State.HOME;
		StateNext(supply_data.state);
	52:
		IF supply_data.axis.state = State.HOME_DONE THEN
			supply_data.state := State.HOME_DONE;
		END_IF
	//////\\
	////\\\\
	//\\\\\\
	State.HOME_OFFSET:
		supply_data.axis.home_offset_micron := 0;
		supply_data.axis.state := State.HOME_OFFSET;
		StateNext(supply_data.state);
	92:
		IF supply_data.axis.state = State.HOME_OFFSET_DONE THEN
			supply_data.axis.state := State.READY;
			supply_data.state := State.HOME_OFFSET_DONE;
		END_IF
	State.READY:
		//do nothing
	//////\\
	////\\\\
	//\\\\\\
	State.RUN:
		supply_data.foil_short := FALSE; // reset giá trị bào hiệu phôi hết
		supply_data.axis.target_velocity_micron_per_sec := supply_data.foil_micron_per_sec;
		supply_data.clamp_hold.on := TRUE; // bật kẹp giữ
		supply_data.clamp_drag.on := TRUE; // bật kẹo kéo
		StateNext(supply_data.state);
	102:
		IF supply_data.clamp_hold.p_timer.Q AND supply_data.clamp_drag.p_timer.Q THEN
			// xem các timer này ở hàm io() 
			StateNext(supply_data.state);
		END_IF
	103:
		supply_data.foil_position_delta_micron := supply_data.foil_position_target_micron - supply_data.foil_position_micron;
		// kiểm tra độ chênh lệch giữa vị trí phôi hiện tại và vị trí phôi mục tiêu
		IF supply_data.foil_position_delta_micron > 0 THEN // nếu > 0 thì cần đẩy phôi
			supply_data.state := 111;
		ELSE // còn <= 0 thì nhảy sang bước 131, nhưng bước này là bước cụt
			supply_data.state := 131;
		END_IF
	//Move foil forward
	111:
		IF supply_data.foil_position_delta_micron > 0 THEN // delta vẫn > 0 thì tiếp tục đẩy
			IF supply_data.foil_position_delta_micron > supply_data.axis.max_micron THEN // nếu delta dài hơn quãng đường có thể chạy của trục
				supply_data.axis.target_position_micron := supply_data.axis.max_micron; // thì chạy tới vị trí max
				supply_data.foil_position_delta_micron := supply_data.foil_position_delta_micron - supply_data.axis.max_micron; // trừ đi max từ delta
			ELSE // nếu bé hơn hoặc bàng max thì đẩy 1 phát nữa là xong
				supply_data.axis.target_position_micron := supply_data.foil_position_delta_micron;
				supply_data.foil_position_delta_micron := 0;
			END_IF
			StateNext(supply_data.state);
		ELSE // delta <= 0 thì xong, phép tính ở trên không thể có kết quả < 0 
			supply_data.foil_position_micron := supply_data.foil_position_target_micron;
			supply_data.state := State.READY;
		END_IF
	112:
		supply_data.clamp_hold.on := TRUE; // bật kẹp giữ
		StateNext(supply_data.state);
	113:
		IF supply_data.clamp_hold.p_timer.Q THEN // p_timer là positive timer, xác định đã bật xylanh sau 1 khoảng thời gian, xem io() và save_apply() 
			supply_data.clamp_drag.on := FALSE;
			StateNext(supply_data.state);
		END_IF
	114:
		IF supply_data.clamp_drag.n_timer.Q AND supply_data.axis.state = State.READY THEN
			supply_data.axis.state := State.RUN;
			StateNext(supply_data.state);
		END_IF
	115:
		IF supply_data.axis.state = State.READY THEN
			IF supply_data.sensor_drag THEN // nếu lúc đi ra để kẹp phôi mà cảm biến còn tín hiệu thì tiếp tục
				supply_data.clamp_drag.on := TRUE;
				StateNext(supply_data.state);
			ELSE // còn không thì dừng ngay tại đây, xem hàm work()
				supply_data.foil_short := TRUE;
				supply_data.state := State.READY;
			END_IF
		END_IF
	116:
		IF supply_data.clamp_drag.p_timer.Q THEN
			supply_data.clamp_hold.on := FALSE;
			StateNext(supply_data.state);
		END_IF
	117:
		IF supply_data.clamp_hold.n_timer.Q AND supply_data.axis.state = State.READY THEN
			supply_data.axis.target_position_micron := 0;
			supply_data.axis.state := State.RUN;
			StateNext(supply_data.state);
		END_IF
	118:
		IF supply_data.axis.state = State.READY THEN
			StateNext(supply_data.state);
		END_IF
	119:
		supply_data.clamp_hold.on := TRUE;
		StateNext(supply_data.state);
	120:
		IF supply_data.clamp_hold.p_timer.Q THEN // kẹp xong quay lại bước 111 để kiểm tra xem đã đẩy hết phôi hay chưa
			supply_data.state := 111;
		END_IF
	//Move foil backward
	131:
		//not implemented yet
END_CASE
END_ACTION

ACTION work:
IF (
	supply_data.axis.overload OR
	cut_data.axis.overload
) THEN
	work_data.overload.on := TRUE;
END_IF

CASE work_data.state OF
	State.RST:
		supply_data.state := State.RST;
		cut_data.state := State.RST;
		StateNext(work_data.state);
	2:
		IF (
			supply_data.state = State.RST_DONE AND
			cut_data.state = State.RST_DONE
		) THEN
			work_data.state := State.RST_DONE;
		END_IF
	State.RST_DONE:
		// do nothing
	//////\\
	////\\\\
	//\\\\\\
	State.HOME:
		supply_data.state := State.HOME;
		cut_data.state := State.HOME;
		StateNext(work_data.state);
	52:
		IF (
			supply_data.state = State.HOME_DONE AND
			cut_data.state = State.HOME_DONE
		) THEN
			work_data.state := State.HOME_DONE;
		END_IF
	State.HOME_DONE:
		supply_data.state := State.HOME_OFFSET;
		cut_data.state := State.HOME_OFFSET;
		StateNext(work_data.state);
	91:
		IF (
			supply_data.state = State.HOME_OFFSET_DONE AND
			cut_data.state = State.HOME_OFFSET_DONE
		) THEN
			work_data.state := State.HOME_OFFSET_DONE;
		END_IF
	State.HOME_OFFSET_DONE:
		supply_data.state := State.READY;
		cut_data.state := State.READY;
		work_data.state := State.READY;
	//////\\
	////\\\\
	//\\\\\\
	State.READY:
		FOR i := 0 TO c_axis_i_max BY 1 DO
			CASE i OF
				0: work_data.jog_i := ADR(supply_data.axis);
				1: work_data.jog_i := ADR(cut_data.axis);
			END_CASE
			work_data.jog_i^.jog_micron_per_sec := hmi_data.jog_micron_per_sec;
			IF hmi_data.jog_n THEN
				work_data.jog_i^.jog_direction := -1;
			END_IF
			IF hmi_data.jog_p THEN
				work_data.jog_i^.jog_direction := +1;
			END_IF
			IF NOT (hmi_data.jog_n OR hmi_data.jog_p) OR i <> hmi_data.jog_index THEN
				work_data.jog_i^.jog_direction := 0;
			END_IF
		END_FOR
	//////\\
	////\\\\
	//\\\\\\
	State.RUN:
		IF cut_data.state = State.READY THEN
			cut_data.state := 151; // kích hoạt lùi dao về begin
			StateNext(work_data.state);
		END_IF
	102:
		IF cut_data.state = State.READY THEN
			work_data.state := 105;
		END_IF
	//phôi tiếp theo
	105:
		work_data.cut_profile := save_data_big.cut_profiles[save_data.cut_profile_index]; // set cut_profile
		work_data.cut_profile_step_index := 0; // set bước cắt trong cut_profile
		supply_data.foil_position_micron := 0; // set vị trí phôi = 0
		supply_data.foil_micron_per_sec := work_data.cut_profile.supply_micron_per_sec;
		cut_data.cut_micron_per_sec := work_data.cut_profile.cut_micron_per_sec;
		work_data.state := 111;
		RTC_last := RTC;
	//CHECK
	111:
		work_data.cut_profile_step := ADR(work_data.cut_profile.steps[work_data.cut_profile_step_index]);
		supply_data.foil_position_target_micron := UDINT_TO_LREAL(work_data.cut_profile_step^.begin_micron);
		IF work_data.cut_profile_step^.active THEN // nếu cut_profile_step được kích hoạt thì nhảy đến bước cắt
			work_data.state := 121;
		ELSE // nếu không thì tiếp tục kiểm tra cut_profile_step tiếp theo
			IF work_data.cut_profile_step_index < c_cut_profile_step_i_max THEN
				work_data.cut_profile_step_index := work_data.cut_profile_step_index + 1;
			ELSE // nếu không còn cut_profile_step nào nữa thì nhảy đến bước 151 để cắt rời
				work_data.state := 151;
			END_IF
		END_IF
	//MIDDLE CUT
	//Calculate
	121:
		// tính vị trí phôi và độ sâu cắt
		// lưu ý: cần đổi số trước khi thực hiện các phép toán có khả năng ảnh hưởng bởi kiểu số
		// ví dụ .depth_end_micron và .depth_begin_micron là kiểu UDINT (unsigned double integer -> số nguyên không âm 32 bit)
		// nếu không đổi sang LREAL (long real -> số thực 64 bit) hay những kiểu dữ liệu hỗ trợ số âm thì sẽ bị tràn
		// nếu .depth_end_micron = 1 và .depth_begin_micron = 2, thì .depth_end_micron - .depth_begin_micron = 1 - 2 = 4_294_967_295
		IF supply_data.foil_position_micron < work_data.cut_profile_step^.begin_micron + work_data.cut_profile_step^.width_micron THEN
			supply_data.foil_position_target_micron := MIN(
				work_data.cut_profile_step^.begin_micron + work_data.cut_profile_step^.width_micron,
				supply_data.foil_position_target_micron + work_data.blade_thickness_micron
			);
			cut_data.depth_micron := work_data.cut_profile_step^.depth_begin_micron;
			cut_data.depth_micron := cut_data.depth_micron + (
				(supply_data.foil_position_target_micron - (UDINT_TO_LREAL(work_data.cut_profile_step^.begin_micron) + work_data.blade_thickness_micron))
				/
				(UDINT_TO_LREAL(work_data.cut_profile_step^.width_micron) - work_data.blade_thickness_micron)
			) * (UDINT_TO_LREAL(work_data.cut_profile_step^.depth_end_micron) - UDINT_TO_LREAL(work_data.cut_profile_step^.depth_begin_micron));
			work_data.state := 131;
		ELSE
			work_data.state := 150;
		END_IF
	//Cut
	131:
		IF supply_data.state = State.READY THEN
			supply_data.state := State.RUN;
			StateNext(work_data.state);
		END_IF
	132:
		IF supply_data.state = State.READY AND NOT supply_data.foil_short THEN // chưa hết phôi thì cắt
			cut_data.state := State.RUN;
			StateNext(work_data.state);
		END_IF
	133:
		IF cut_data.state = State.READY THEN
			work_data.state := 121;
		END_IF
	//Return or end
	150:
		IF work_data.cut_profile_step_index < c_cut_profile_step_i_max THEN
			work_data.cut_profile_step_index := work_data.cut_profile_step_index + 1;
			work_data.state := 111;
		ELSE
			work_data.state := 151;
		END_IF
	//TAIL CUT
	151:
		IF supply_data.state = State.READY THEN
			supply_data.foil_position_target_micron := work_data.cut_profile.length_micron + work_data.blade_thickness_micron;
			supply_data.state := State.RUN;
			StateNext(work_data.state);
		END_IF
	152:
		IF supply_data.state = State.READY AND NOT supply_data.foil_short THEN // chưa hết phôi thì cắt
			cut_data.depth_micron := work_data.cut_depth_end_micron;
			cut_data.state := State.RUN;
			StateNext(work_data.state);
		END_IF
	153:
		IF cut_data.state = State.READY THEN
			work_data.work_piece_remain := work_data.work_piece_remain - 1; // số phôi cần cắt còn lại -1
			IF work_data.work_piece_remain > 0 THEN
				work_data.state := 105; // nhảy đến bước phôi tiếp theo
			ELSE
				work_data.state := State.READY;
				hmi_data.view_cycle_time_msec := ULINT_TO_UDINT(RTC - RTC_last); // tính thời gian cắt, xem bước RUN ở trên
			END_IF
		END_IF
	//////\\
	////\\\\
	//\\\\\\
	171: // cắt thử công, xem chương trình kích hoạt trong hàm io()
		IF cut_data.state = State.READY THEN
			cut_data.depth_micron := work_data.cut_depth_end_micron;
			cut_data.cut_micron_per_sec := work_data.manual_cut_micron_per_sec;
			cut_data.state := State.RUN;
			StateNext(work_data.state);
		END_IF
	172:
		IF cut_data.state = State.READY THEN
			work_data.state := State.READY;
		END_IF
END_CASE
END_ACTION

ACTION cut:
////////
//MAIN//
////////
cut_data.axis_fb(data:= ); // data của hàm này đã được set ở hàm MAIN
CASE cut_data.state OF
	//////\\
	////\\\\
	//\\\\\\
	State.RST:
		cut_data.axis.state := State.RST;
		StateNext(cut_data.state);
	2:
		IF cut_data.axis.state = State.RST_DONE THEN
			cut_data.state := State.RST_DONE;
		END_IF
	//////\\
	////\\\\
	//\\\\\\
	State.HOME:
		cut_data.axis.state := State.HOME;
		StateNext(cut_data.state);
	52:
		IF cut_data.axis.state = State.HOME_DONE THEN
			cut_data.state := State.HOME_DONE;
		END_IF
	//////\\
	////\\\\
	//\\\\\\
	State.HOME_OFFSET:
		cut_data.axis.home_offset_micron := 0;
		cut_data.axis.state := State.HOME_OFFSET;
		StateNext(cut_data.state);
	92:
		IF cut_data.axis.state = State.HOME_OFFSET_DONE THEN
			cut_data.axis.state := State.READY;
			cut_data.state := State.HOME_OFFSET_DONE;
		END_IF
	//////\\
	////\\\\
	//\\\\\\
	State.READY:
		//do nothing
	//////\\
	////\\\\
	//\\\\\\
	State.RUN:
		IF cut_data.axis.state = State.READY THEN
			cut_data.axis.target_position_micron := cut_data.begin_micron;
			cut_data.axis.target_velocity_micron_per_sec := cut_data.cut_retract_micron_per_sec;
			cut_data.axis.state := State.RUN;
			StateNext(cut_data.state);
		END_IF
	102:
		IF cut_data.axis.state = State.READY THEN
			cut_data.axis.target_position_micron := cut_data.begin_micron + cut_data.depth_micron; // đã có giới hạn trong AxisLinearFB nên không cần giới hạn ở đây
			cut_data.axis.target_velocity_micron_per_sec := cut_data.cut_micron_per_sec;
			cut_data.axis.state := State.RUN;
			StateNext(cut_data.state);
		END_IF
	103:
		IF cut_data.axis.state = State.READY THEN
			cut_data.axis.target_position_micron := cut_data.begin_micron;
			cut_data.axis.target_velocity_micron_per_sec := cut_data.cut_retract_micron_per_sec;
			cut_data.axis.state := State.RUN;
			StateNext(cut_data.state);
		END_IF
	104:
		IF cut_data.axis.state = State.READY THEN
			cut_data.state := State.READY;
		END_IF
	//////\\
	////\\\\
	//\\\\\\
	151: // lùi dao về 0
		IF cut_data.axis.state = State.READY THEN
			cut_data.axis.target_position_micron := cut_data.begin_micron;
			cut_data.axis.target_velocity_micron_per_sec := cut_data.cut_retract_micron_per_sec;
			cut_data.axis.state := State.RUN;
			StateNext(cut_data.state);
		END_IF
	152:
		IF cut_data.axis.state = State.READY THEN
			cut_data.state := State.READY;
		END_IF
END_CASE
END_ACTION

ACTION cut_profile_update:
process_data.cut_profile_name := save_data.cut_profiles_name[hmi_data.save_data.cut_profile_index];
MEMUtils.MemCpy(
	ADR(hmi_data.cut_profile_name_as_array),
	ADR(process_data.cut_profile_name),
	UINT_TO_DWORD(c_name_length)
);
// đây là hàm vẽ hình
// .cut_profile_points_x và .cut_profile_points_y là 2 mảng dùng để lưu vị trí cho HMI vẽ ra cut_profile
// với 5 step, mỗi step 4 điểm cộng với 2 điểm đầu và 2 điểm cuối ta có mảng gồm 24 phần tử
// hình vẽ có gốc toạ độ ở phía trên, bên trái

hmi_data.cut_profile := save_data_big.cut_profiles[hmi_data.save_data.cut_profile_index];
hmi_data.cut_profile_point_count := 2; // 2 điểm đầu tiên là điểm (0, max_depth) và điểm (0, 0)
hmi_data.cut_profile_points_x[0] := 0;
hmi_data.cut_profile_points_y[0] := LREAL_TO_UDINT(cut_data.axis.max_micron);
hmi_data.cut_profile_points_x[1] := 0;
hmi_data.cut_profile_points_y[1] := 0;
FOR i := 0 TO c_cut_profile_step_i_max BY 1 DO
	cut_profile_step_i := ADR(hmi_data.cut_profile.steps[i]);
	IF cut_profile_step_i^.active THEN
		// nếu cut_profile_step.active = TRUE
		// mỗi cut_profile_step cần vẽ 4 điểm
		j := hmi_data.cut_profile_point_count;
		//
		hmi_data.cut_profile_points_x[j] := MAX(0, cut_profile_step_i^.begin_micron - save_data.blade_thickness_micron);
		hmi_data.cut_profile_points_y[j] := 0;
		hmi_data.cut_profile_points_x[j+1] := hmi_data.cut_profile_points_x[j];
		hmi_data.cut_profile_points_y[j+1] := cut_profile_step_i^.depth_begin_micron;
		//
		hmi_data.cut_profile_points_x[j+2] := cut_profile_step_i^.begin_micron + cut_profile_step_i^.width_micron;
		hmi_data.cut_profile_points_y[j+2] := cut_profile_step_i^.depth_end_micron;
		hmi_data.cut_profile_points_x[j+3] := hmi_data.cut_profile_points_x[j+2];
		hmi_data.cut_profile_points_y[j+3] := 0;
		//
		hmi_data.cut_profile_point_count := hmi_data.cut_profile_point_count + 4; // +4 điểm vào point_count
	END_IF
END_FOR
j := hmi_data.cut_profile_point_count;
hmi_data.cut_profile_points_x[j] := hmi_data.cut_profile.length_micron;
hmi_data.cut_profile_points_y[j] := 0;
hmi_data.cut_profile_points_x[j+1] := hmi_data.cut_profile_points_x[j];
hmi_data.cut_profile_points_y[j+1] := hmi_data.cut_profile_points_y[0];
hmi_data.cut_profile_point_count := hmi_data.cut_profile_point_count + 2; // 2 điểm cuối là (length, 0) và (length, max_depth)
//
// bound là một hình hộp chữ nhật bao lấy cut_profile
hmi_data.cut_profile_bound_x := hmi_data.cut_profile.length_micron; // bound_x là độ rộng
hmi_data.cut_profile_bound_y := hmi_data.cut_profile_points_y[0] - save_data.cut_begin_micron; // bound_y là độ cao
// bound_x và bound_y dùng để hỗ trợ tính toán trên HMI
// ví dụ bound_x = 1000_000, bound_y = 150_000, trong khi khung vẽ trên HMI có độ phân giải là 780x180
// cần phải có bound để HMI tình toán độ phóng to thu nhỏ
// xem macro cut_profile_update() trên HMI để biết thêm chi tiết
END_ACTION

END_PROGRAM

// Device/Application/StateNext
FUNCTION StateNext
VAR_INPUT
	state: REFERENCE TO INT;
END_VAR
VAR
END_VAR

state := state + 1;

END_FUNCTION

// Device/Application/AxisLinearFB
FUNCTION_BLOCK PUBLIC AxisLinearFB
VAR_INPUT
	data: POINTER TO AxisLinear;
END_VAR
VAR_OUTPUT
END_VAR
VAR
END_VAR

data^.torque_Nm := data^.ref^.fActTorque * 1E-3 * data^.torque_rated_Nm;
// giá trị .fActTorque có thể khác nhau tuỳ PLC, trong trường hợp PLC Inovance này fActTorque là giá trị từ phần trăm moment
// 0.0% đến hơn 100.0%, nên phải nhân với .torque_rated_Nm đọc được ở hàm MAIN
data^.home_hit_timer(IN:= , PT:= , Q=> , ET=> );
// timer để lấy gốc, khi lùi về chạm gốc, giá trị moment sẽ tăng lên đến giá trị quy định (trong chương trình này là 1.27Nm)
// để tránh bị nhiễu thì moment quy định cần phải duy trì trong một thời gian mới có thể xác định gốc
data^.overload_timer(IN:= , PT:= , Q=> , ET=> );
// timer quá tải
IF data^.state >= State.READY THEN
	data^.overload_timer.IN := data^.torque_Nm > (1.0 * data^.torque_rated_Nm);
	data^.overload := data^.overload_timer.Q OR data^.torque_Nm > (3.0 * data^.torque_rated_Nm);
END_IF
//////\\
////\\\\
//\\\\\\
CASE data^.state OF
	State.RST: // reset trục
		data^.read_status^.Enable := TRUE; // bật đọc trạng thái servo
		StateNext(data^.state);
	2:
		IF data^.read_status^.Valid THEN
			StateNext(data^.state);
		END_IF
	3:
		data^.inch^.InchBackward := FALSE;
		data^.inch^.InchForward := FALSE;
		IF data^.mabs^.Busy THEN // nếu hàm dịch chuyển MC_MoveAbsolute đang hoạt dộng thì kích hoạt hàm MC_Stop
			data^.stop^.Deceleration := data^.mabs^.Velocity / 0.1;
			data^.stop^.Jerk := data^.stop^.Deceleration * data^.jerk_factor;
			data^.stop^.Execute := TRUE;
			StateNext(data^.state);
		ELSE // nếu không thì nhảy đến bước tiếp theo
			data^.state := 21;
		END_IF
	4: // hàm SMC_Inch đang không hoạt động và hàm MC_Stop hoàn thành
		IF NOT data^.inch^.Busy AND data^.stop^.Done THEN
			data^.state := 21;
		END_IF
	//
	21:
		data^.mabs^.Execute := FALSE; // sau khi các hàm hoàn thành, phải đặt biến Execute về FALSE
		data^.stop^.Execute := FALSE; // vì muốn chạy hàm cần có tín hiệu rising edge
		data^.power^.bDriveStart := FALSE; // tắt servo
		StateNext(data^.state);
	22:
		IF NOT data^.power^.Status THEN // đã tắt xong servo
			StateNext(data^.state);
		END_IF
	23:
		IF data^.read_status^.FBErrorOccured THEN // nếu có lỗi xảy ra thì xoá lỗi cũ
			SMC_ClearFBError(pDrive:= data^.ref); // xoá lỗi
			StateNext(data^.state);
		ELSE // nếu không có thì nhảy đến bước cuối
			data^.state := 31;
		END_IF
	24:
		IF data^.read_status^.FBErrorOccured THEN
			data^.reset^.Execute := TRUE; // reset lỗi
			StateNext(data^.state);
		END_IF
	25:
		IF data^.reset^.Done THEN
			data^.reset^.Execute := FALSE;
			SMC_ClearFBError(pDrive:= data^.ref); // xoá lỗi
			data^.state := 31;
		END_IF
	//
	31:
		data^.read_status^.Enable := FALSE;
		data^.state := State.RST_DONE;
	//////\\
	////\\\\
	//\\\\\\
	State.HOME:
		data^.power^.bDriveStart := TRUE; // bật servo để bắt đầu lấy gốc
		StateNext(data^.state);
	52:
		IF data^.power^.Status THEN // servo đã sẵn sàng
			StateNext(data^.state);
		END_IF
	53:
		IF data^.home_done THEN // đã lấy gốc trước đó thì nhảy đến bước HOME_FORWARD
			data^.state := State.HOME_FORWARD;
		ELSE // chưa lấy gốc thì qua bước tiếp theo
			StateNext(data^.state);
		END_IF
	54:
		data^.set_mode^.nControllerMode := SMC_CONTROLLER_MODE.SMC_velocity;// chuyển chế độ servo sang tốc độ
		// ở chế độ .SMC_torque hoặc .SMC_velocity, khi servo vị chặn nó sẽ không vọt sau khi được nhả ra
		data^.set_mode^.bExecute := TRUE;
		StateNext(data^.state);
	55:
		IF data^.set_mode^.bDone THEN // chuyển chế độ xong
			data^.set_mode^.bExecute := FALSE;
			StateNext(data^.state);
		END_IF
	56:
		data^.home_torque_Nm := MIN(1.27, data^.torque_rated_Nm);
		// đặt giá trị moment, 1.27Nm là tối đa, với vít me bước 5mm thì lực ép ở 1.27Nm sẽ là (1.27*2*PI)/0.005 = 1595N
		// khoảng 160 kg
		// moment không được vượt quá moment danh định vì nó sẽ lỗi quá tải khi ngâm ở thời gian dài với home_hit_timer
		data^.limit_torque^.NegativeEnable := TRUE;
		data^.limit_torque^.PositiveEnable := TRUE;
		data^.limit_torque^.NegativeValue := 1000 * (data^.home_torque_Nm / data^.torque_rated_Nm);
		data^.limit_torque^.PositiveValue := 1000 * (data^.home_torque_Nm / data^.torque_rated_Nm);
		data^.limit_torque^.Execute := TRUE;
		// thực thi hàm limit_torque
		// hãy đọc function defination của hàm này
		// giá trị 1000 tức là 100% moment vì step là 0.1% mỗi đơn vị
		StateNext(data^.state);
	57:
		IF data^.limit_torque^.Done THEN // set xong giới hạn moment
			data^.limit_torque^.Execute := FALSE;
			StateNext(data^.state);
		END_IF
	58:
		data^.inch^.Velocity := data^.home_back_micron_per_sec; // lùi về
		data^.inch^.Distance := 500_000; // hàm SMC_Inch có giới hạn bới .Distance, khác với hàm MC_Jog không có giới hạn
		// đặt .Distance = 500_000 hay số nào đó thật lớn cũng được
		data^.inch^.Acceleration := data^.inch^.Velocity / 0.1;
		data^.inch^.Deceleration := data^.inch^.Acceleration;
		data^.inch^.Jerk := data^.inch^.Acceleration * data^.jerk_factor;
		data^.inch^.InchBackward := TRUE; // .InchBackward là lùi
		data^.inch^.InchForward := FALSE; // .InchForward là tiến
		// nếu .InchBackward và .InchForward cùng bằng TRUE hoặc FALSE thì servo không chạy
		data^.home_hit_timer.IN := FALSE; // reset timer
		StateNext(data^.state);
	59:
		data^.home_hit_timer.IN := ABS(data^.torque_Nm) >= data^.home_torque_Nm * 0.95; // set timer, * 0.95 để chắc ăn, tránh bị nhiễu
		IF data^.home_hit_timer.Q THEN // khi timer kích hoạt, dừng hàm SMC_Inch
			data^.inch^.InchBackward := FALSE;
			data^.inch^.InchForward := FALSE;
			data^.mabs^.Position := data^.ref^.fActPosition + data^.home_offset_absolute_micron;
			// gán tạm giá trị vào hàm MC_MoveAbsolute để đến bước tiếp theo
			// .fActPosition là vị trí thực tế của servo
			// ví dụ .fActPosition khi chạm là -123_000, có thể dùng "_" để phân cách các con số cho dễ đọc
			// .home_offset_absolute_micron = 1_000
			// data^.mabs^.Position sẽ bằng -123_000 + 1_000 = -122_000
			StateNext(data^.state);
		END_IF
	60:
		data^.sp^.Position := data^.ref^.fActPosition - data^.mabs^.Position;
		// thực hiện hàm MC_SetPosition để đưa giá trị .fActPosition về 0
		// bây giờ giá trị data^.sp^.Position = -123_000 - (-122_000) = -1_000
		// bây giờ servo đang ở vị trí va chạm, để về gốc thì nó phải dịch chuyển 1_000 micron
		// vậy vị trí gốc cách vị trí va chạm đúng bằng .home_offset_absolute_micron
		data^.sp^.Execute := TRUE;
		StateNext(data^.state);
	61:
		IF data^.sp^.Done THEN // set xong tiến tới HOME_FORWARD
			data^.sp^.Execute := FALSE;
			data^.state := State.HOME_FORWARD;
			data^.home_done := TRUE;
		END_IF
	//////\\
	////\\\\
	//\\\\\\
	State.HOME_FORWARD:
		IF NOT data^.inch^.Busy THEN
			data^.set_mode^.nControllerMode := SMC_CONTROLLER_MODE.SMC_position; // set mode về điều khiển vị trí
			data^.set_mode^.bExecute := TRUE;
			StateNext(data^.state);
		END_IF
	72:
		IF data^.set_mode^.bDone THEN
			data^.set_mode^.bExecute := FALSE;
			StateNext(data^.state);
		END_IF
	73:
		data^.limit_torque^.NegativeEnable := TRUE;
		data^.limit_torque^.PositiveEnable := TRUE;
		data^.limit_torque^.NegativeValue := 3000;
		data^.limit_torque^.PositiveValue := 3000;
		data^.limit_torque^.Execute := TRUE;
		StateNext(data^.state);
		// đưa giới hạn moment về 300%
	74:
		IF data^.limit_torque^.Done THEN
			data^.limit_torque^.Execute := FALSE;
			StateNext(data^.state);
		END_IF
	75:
		// dịch chuyển tới vị trí gốc
		data^.mabs^.Position := 0;
		data^.mabs^.Velocity := data^.home_forward_micron_per_sec;
		data^.mabs^.Acceleration := data^.mabs^.Velocity / data^.ramp_time_sec;
		data^.mabs^.Deceleration := data^.mabs^.Acceleration;
		data^.mabs^.Jerk := data^.mabs^.Acceleration * data^.jerk_factor;
		data^.mabs^.Execute := TRUE;
		StateNext(data^.state);
	76:
		IF data^.mabs^.Done THEN
			data^.mabs^.Execute := FALSE;
			data^.state := State.HOME_DONE;
		END_IF
	//////\\
	////\\\\
	//\\\\\\
	State.HOME_OFFSET: // địch chuyển tới vị trí HOME_OFFSET
		data^.mabs^.Position := data^.home_offset_micron;
		data^.mabs^.Velocity := data^.home_forward_micron_per_sec;
		data^.mabs^.Acceleration := data^.mabs^.Velocity / data^.ramp_time_sec;
		data^.mabs^.Deceleration := data^.mabs^.Acceleration;
		data^.mabs^.Jerk := data^.mabs^.Acceleration * data^.jerk_factor; // jerk chỉ có tác dụng khi Velocity ramp type khác Trapezoid
		data^.mabs^.Execute := TRUE;
		StateNext(data^.state);
	92:
		IF data^.mabs^.Done THEN // dịch chuyển xong
			data^.mabs^.Execute := FALSE;
			data^.state := State.HOME_OFFSET_DONE;
		END_IF
	//////\\
	////\\\\
	//\\\\\\
	State.READY:
		// trạng thái sẵn sàng đợi lệnh, có thể jog
		// hàm SMC_Inch có giới hạn .Distance
		// ta dùng giới hạn này để giới hạn hành trình jog, tránh va chạm
		data^.inch^.Velocity := data^.jog_micron_per_sec;
		data^.inch^.Acceleration := data^.inch^.Velocity / data^.ramp_time_sec;
		data^.inch^.Deceleration := data^.inch^.Acceleration;
		data^.inch^.Jerk := data^.inch^.Acceleration * data^.jerk_factor;
		data^.inch^.InchBackward := data^.jog_direction = -1;
		data^.inch^.InchForward := data^.jog_direction = +1;
		IF data^.inch^.InchBackward THEN
			data^.inch^.Distance := data^.ref^.fActPosition;
			// khi đi lùi, ví dụ servo ở vị trí 12_000
			// .Distance bằng 12_000
		END_IF
		IF data^.inch^.InchForward THEN
			data^.inch^.Distance := data^.max_micron - data^.ref^.fActPosition;
			// khi tiến, ví dụ hành trình tối đa là 155_000
			// vị trí hiện tại là 100_000
			// .Distance bằng 155_000 - 100_000 = 55_000
		END_IF
	//////\\
	////\\\\
	//\\\\\\
	State.RUN:
		// lệnh chạy đến vị trí chỉ định
		// xem hàm cut() và supply()
		// set data^.target_position_micron và data^.target_velocity_micron_per_sec sau đó set data^.state = State.RUN
		data^.mabs^.Position := MAX(0, MIN(data^.max_micron, data^.target_position_micron)); // giới hạn vị trí, xem save_apply()
		data^.mabs^.Velocity := MAX(0_100, MIN(data^.max_micron_per_sec, data^.target_velocity_micron_per_sec)); // giới hạn tốc độ, xem save_apply()
		data^.mabs^.Acceleration := data^.mabs^.Velocity / data^.ramp_time_sec;
		data^.mabs^.Deceleration := data^.mabs^.Acceleration;
		data^.mabs^.Jerk := data^.mabs^.Acceleration * data^.jerk_factor;
		data^.mabs^.Execute := TRUE;
		StateNext(data^.state);
	102:
		IF data^.mabs^.Done THEN
			data^.mabs^.Execute := FALSE;
			data^.state := State.READY;
		END_IF
END_CASE

END_FUNCTION_BLOCK
